{attribute 'GeneratedUsingTerminal: EL2521-0124-0018'}
{attribute addProperty BoxType "EL2521-0124-0018"}
{attribute addProperty Id "StatusAT %I*Status_7097155E4"}
{attribute addProperty CRC "1894228450"}
{attribute addProperty Size "4"}
TYPE PLS_Status_70E7A1E2 :
STRUCT
	{attribute addProperty Name "Status"}
	Status AT %I* : Status_7097155E;
END_STRUCT
END_TYPE

(* stored: Version 1.2.0.0, ProductVersion 3.1.4024.9
   DUT PLS_Status_70E7A1E2: Id {93ee0436-2f87-4793-8d45-b7ee252cba72} *)
